// TwinCAT 3 PLC project PorjectPanel
// ProgramVersion: 3.1.4026.1+c9eadab3edd020c56c333d811d5b3c408c2550c8
// libraries:
//   Tc2_Standard, * (Beckhoff Automation GmbH)
//   Tc2_System, * (Beckhoff Automation GmbH)
// project tree:
//   GVLs/ gProjectHpuIO.TcGVL
//   / PlcTask.TcTTO (not stored)
//   POUs/ MAIN.TcPOU
// real-time tasks:
//   TASK PlcTask: cycle T#10ms, priority 20, ADS port 350
// variable links:
//   HPU Instance <-> ProjectPanel/ProjectPanel Instance
//     PlcTask Inputs/gHpuProjectIO.heatRequest <-> PlcTask Outputs/gProjectHpuIO.heatRequest
//     PlcTask Inputs/gHpuProjectIO.hoFlow <-> PlcTask Outputs/gProjectHpuIO.hoFlow
//     PlcTask Outputs/gHpuProjectIO.heater1Status <-> PlcTask Inputs/gProjectHpuIO.heater1Status
//     PlcTask Outputs/gHpuProjectIO.powerAvailable <-> PlcTask Inputs/gProjectHpuIO.powerAvailable

// ---- GVLs/gProjectHpuIO.TcGVL
{attribute 'qualified_only'}
VAR_GLOBAL
	heatRequest		AT %Q*	: BOOL;
	powerAvailable	AT %I*	: REAL;
	
	heater1Status	AT %I*	: BOOL;
	hoFlow			AT %Q*	: REAL;	
	
END_VAR

// ---- POUs/MAIN.TcPOU
PROGRAM MAIN
VAR
END_VAR

END_PROGRAM
